// Mitsubishi GX Works2 project: PLC   PLC: FX3G

PROGRAM MAIN
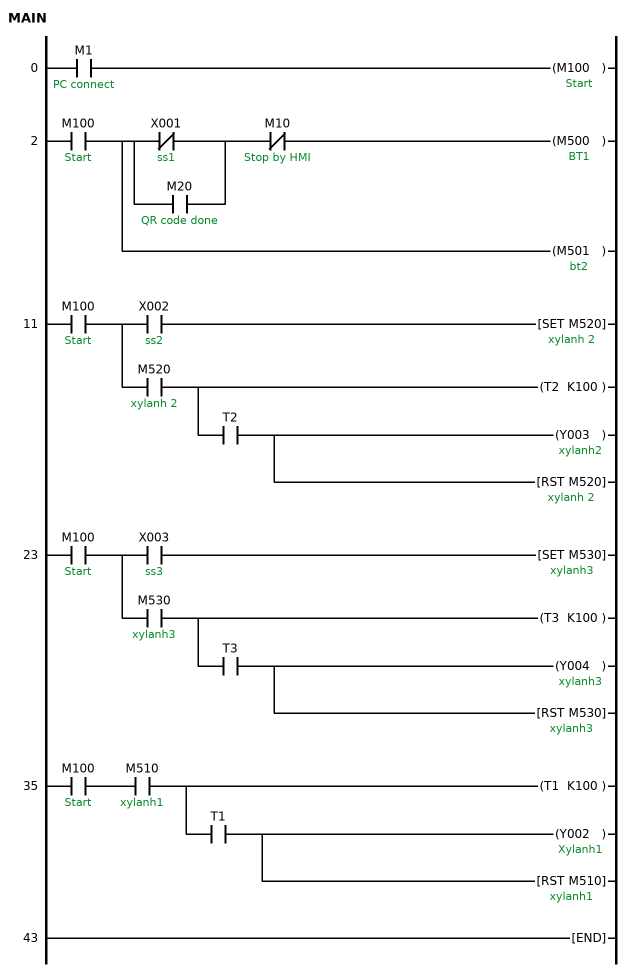
0     LD      M1  ; PC connect
      OUT     M100  ; Start
2     LD      M100  ; Start
      MPS
      LDI     X001  ; ss1
      OR      M20  ; QR code done
      ANB
      ANI     M10  ; Stop by HMI
      OUT     M500  ; BT1
      MPP
      OUT     M501  ; bt2
11    LD      M100  ; Start
      MPS
      AND     X002  ; ss2
      SET     M520  ; xylanh 2
      MPP
      AND     M520  ; xylanh 2
      OUT     T2 K100
      AND     T2
      OUT     Y003  ; xylanh2
      RST     M520  ; xylanh 2
23    LD      M100  ; Start
      MPS
      AND     X003  ; ss3
      SET     M530  ; xylanh3
      MPP
      AND     M530  ; xylanh3
      OUT     T3 K100
      AND     T3
      OUT     Y004  ; xylanh3
      RST     M530  ; xylanh3
35    LD      M100  ; Start
      AND     M510  ; xylanh1
      OUT     T1 K100
      AND     T1
      OUT     Y002  ; Xylanh1
      RST     M510  ; xylanh1
43    END
END_PROGRAM
